// TIA Portal V18 export
// export: Created 2026-06-08T17:01:58.0454225Z, ExportSetting WithDefaults, DisplayName Totally Integrated Automation Portal, DisplayVersion V18, DisplayName TIA Portal Openness, DisplayVersion V18, DisplayName TIA Portal Version Control Interface, DisplayVersion V18, DisplayName STEP 7 Professional, DisplayVersion V18, DisplayName STEP 7 Safety, DisplayVersion V18, DisplayName WinCC Professional, DisplayVersion V18
DATA_BLOCK "MAIN_I/O_DB"   // DB1
{ S7_Optimized_Access := 'FALSE' }
VERSION : 0.1
// stored: AutoNumber true, DBAccessibleFromOPCUA true, IsOnlyStoredInLoadMemory false, IsWriteProtectedInAS false
   VAR
      MAIN_MOVE_R : Bool;
      MAIN_MOVE_F : Bool;
      MAIN_STOP : Bool;
      SENSOR_HOME : Bool;
      SENSOR_FINISH_1 : Bool;
      SENSOR_FINISH_2 : Bool;
      EMERGENCY : Bool;
      RESET : Bool;
      MAIN_COIL_F : Bool;
      MAIN_COIL_R : Bool;
      COIL_EMERGENCY : Bool;
   END_VAR
BEGIN
END_DATA_BLOCK
